Staubli VAL3: pp_bs_f2f3.pgx

program pp_bs_f2f3()
begin
  //given f2,f3 are in hand
  //exit state : f2, f3 secured in one hand

  //place f2 in origin of bk (//open bk vacuum
  call regular_place(t2,mNomSpeed,mSlowSpeed,pPointRx_f2_bk,false,dDio_t2_cy,true)

  //drop f3 offset from f2 origin
  call regular_pick(t3,mNomSpeed,mSlowSpeed,pPointRx_f3_bk,dDio_t3_cy,false,dDio_f3_secure)

end
